FUNCTION_BLOCK SimpleModel (* Composite Function Block Type *)
  (* Standard: 61499-2 *)
  (* Version 0.0, 6/17/2016, Andrei, nxtControl GmbH, template *)
  PACKAGE Main;
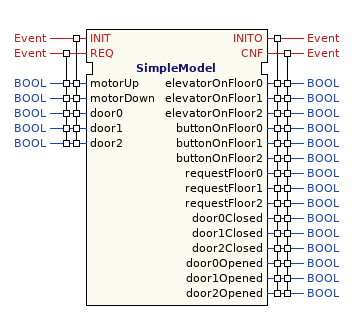
  EVENT_INPUT
    INIT WITH motorUp, motorDown, door0, door1, door2; (* Initialization Request *)
    REQ WITH motorUp, motorDown, door0, door1, door2; (* Normal Execution Request *)
  END_EVENT
  EVENT_OUTPUT
    INITO WITH buttonOnFloor0, buttonOnFloor1, buttonOnFloor2, requestFloor0, requestFloor1, requestFloor2, elevatorOnFloor0, elevatorOnFloor1, elevatorOnFloor2, door0Closed, door1Closed, door2Closed, door0Opened, door1Opened, door2Opened; (* Initialization Confirm *)
    CNF WITH buttonOnFloor0, buttonOnFloor1, buttonOnFloor2, requestFloor0, requestFloor1, requestFloor2, elevatorOnFloor0, elevatorOnFloor1, elevatorOnFloor2, door0Closed, door1Closed, door2Closed, door0Opened, door1Opened, door2Opened; (* Execution Confirmation *)
  END_EVENT
  VAR_INPUT
    motorUp : BOOL; (* Input event qualifier *)
    motorDown : BOOL;
    door0 : BOOL;
    door1 : BOOL;
    door2 : BOOL;
  END_VAR
  VAR_OUTPUT
    elevatorOnFloor0 : BOOL;
    elevatorOnFloor1 : BOOL;
    elevatorOnFloor2 : BOOL;
    buttonOnFloor0 : BOOL; (* Output event qualifier *)
    buttonOnFloor1 : BOOL;
    buttonOnFloor2 : BOOL;
    requestFloor0 : BOOL;
    requestFloor1 : BOOL;
    requestFloor2 : BOOL;
    door0Closed : BOOL;
    door1Closed : BOOL;
    door2Closed : BOOL;
    door0Opened : BOOL;
    door1Opened : BOOL;
    door2Opened : BOOL;
  END_VAR
  FBS
    FB1 : Lift;
    FB2 : FloorIndicator;
    FB3 : ReqPanelLift;
    FB8 : E_MERGE;
    Door0 : Door;
    Door1 : Door;
    Door2 : Door;
    Button0 : CallButton;
    Button1 : CallButton;
    Button2 : CallButton;
    FB5 : MergeEvents;
    FB6 : MergeEvents;
    FB7 : FloorSensors;
    FB4 : Interlock;
    FB9 : ResetDetect;
  END_FBS
  EVENT_CONNECTIONS
    REQ TO FB1.REQ;
    INIT TO FB1.INIT;
    FB1.CNF TO FB7.REQ;
    FB1.INITO TO Door0.INIT;
    Door0.INITO TO Door1.INIT;
    Door1.INITO TO Door2.INIT;
    Door2.INITO TO Button2.INIT;
    Button2.INITO TO Button1.INIT;
    Button1.INITO TO Button0.INIT;
    Button0.INITO TO FB3.INIT;
    FB3.INITO TO INITO;
    FB7.CNF TO FB2.REQ;
    FB1.INITO TO FB2.INIT;
    FB8.EO TO CNF;
    Door0.CNF TO FB5.EI2;
    Door1.CNF TO FB5.EI3;
    Door2.CNF TO FB5.EI4;
    FB3.CNF TO FB6.EI1;
    Button0.CNF TO FB6.EI2;
    Button1.CNF TO FB6.EI3;
    Button2.CNF TO FB6.EI4;
    FB6.EO TO FB8.EI2;
    FB5.EO TO FB8.EI1;
    FB1.CNF TO Door1.REQ;
    FB1.CNF TO Door2.REQ;
    FB1.CNF TO Door0.REQ;
    REQ TO FB3.REQ;
    REQ TO Button0.REQ;
    REQ TO Button1.REQ;
    REQ TO Button2.REQ;
    FB7.CNF TO FB5.EI1;
    FB4.CNF TO FB3.REQ;
    FB4.CNF TO Button0.REQ;
    FB4.CNF TO Button1.REQ;
    FB4.CNF TO Button2.REQ;
    FB6.EO TO FB4.REQ;
    FB7.CNF TO FB9.REQ;
    Door0.CNF TO FB9.REQ;
    Door1.CNF TO FB9.REQ;
    FB9.RST TO FB4.RESET;
    FB5.EO TO FB9.REQ;
  END_CONNECTIONS
  DATA_CONNECTIONS
    motorUp TO FB1.MoveUp;
    motorDown TO FB1.MoveDown;
    FB4.L1 TO requestFloor0;
    FB4.L3 TO requestFloor2;
    FB1.LiftPos TO FB7.CarPos;
    FB7.CarAt2 TO elevatorOnFloor2;
    FB7.CarAt1 TO elevatorOnFloor1;
    FB7.CarAt0 TO elevatorOnFloor0;
    Door0.DoorClosed TO door0Closed;
    door0 TO Door0.OpenDoor;
    door1 TO Door1.OpenDoor;
    door2 TO Door2.OpenDoor;
    Door1.DoorClosed TO door1Closed;
    Door2.DoorClosed TO door2Closed;
    FB4.L4 TO buttonOnFloor0;
    FB4.L5 TO buttonOnFloor1;
    FB4.L6 TO buttonOnFloor2;
    FB7.CarAtFloor TO FB2.FloorNumber;
    Door2.DoorOpened TO door2Opened;
    Door1.DoorOpened TO door1Opened;
    Door0.DoorOpened TO door0Opened;
    FB3.ButtonFor0 TO FB4.B1;
    FB3.ButtonFor1 TO FB4.B2;
    FB3.ButtonFor2 TO FB4.B3;
    Button0.ButtonPressed TO FB4.B4;
    Button1.ButtonPressed TO FB4.B5;
    Button2.ButtonPressed TO FB4.B6;
    FB4.L5 TO Button1.LightON;
    FB4.L6 TO Button2.LightON;
    FB4.L4 TO Button0.LightON;
    FB4.L1 TO FB3.LightON0;
    FB4.L2 TO FB3.LightON1;
    FB4.L3 TO FB3.LightON2;
    FB7.CarAt0 TO FB9.At0;
    FB7.CarAt1 TO FB9.At1;
    FB7.CarAt2 TO FB9.At2;
    Door0.DoorOpened TO FB9.Open0;
    Door1.DoorOpened TO FB9.Open1;
    Door2.DoorOpened TO FB9.Open2;
    FB4.L2 TO requestFloor1;
  END_CONNECTIONS
END_FUNCTION_BLOCK
